// TIA Portal project "weight-based-product-sorting-system" (V16)
// Vorlageprojekt für das Buch mit Zielsystem S7-1200

(* hardware
DEVICE "S7-1200-Station_1"  S7-1200 Station
   slot 0: "Baugruppenträger_0"  Rack  V1.0
   slot 1: "PLC_1"  CPU 1214C DC/DC/DC  6ES7 214-1AG40-0XB0  V4.4
   slot 2: "AQ 4x14BIT_1"  6ES7 232-4HD32-0XB0  V2.1
*)

// ===== PLC "PLC_1"  CPU 1214C DC/DC/DC =====

VAR_GLOBAL   // PLC tag table "Standard-Variablentabelle"
   "Start" AT %I0.0 : Bool;
   "Stop" AT %I0.1 : Bool;
   "Konveyör_Hız_Ayar" AT %IW10 : Int;
   "Giriş_Konveyör" AT %QW20 : Int;
   "Reset_But" AT %I0.2 : Bool;
   "Acil_Stop_But" AT %I0.3 : Bool;
   "Kantar_Giriş_Sensörü" AT %I0.4 : Bool;
   "Kantar_Sensörü" AT %I0.5 : Bool;
   "Kantar_Konveyörü_İleri" AT %Q0.0 : Bool;
   "Ağırlık" AT %IW12 : Int;
   "Transferde_Sensörü" AT %I0.6 : Bool;
   "İleri_Transfer_Konveyörü" AT %Q0.1 : Bool;
   "Ağırlık_Gösterge" AT %QW22 : Int;
   "Sola_Sensör" AT %I0.7 : Bool;
   "Sağa_Sensör" AT %I1.0 : Bool;
   "Sola_Çıkış_Sensörü" AT %I1.1 : Bool;
   "Sağa_Çıkış_Sensörü" AT %I1.2 : Bool;
   "Sağ_Kutu_Sensörü" AT %I1.3 : Bool;
   "Sol_Kutu_Sensörü" AT %I1.4 : Bool;
   "Sol_Konveyör_1" AT %QW24 : Int;
   "Sol_Konveyör_2" AT %Q0.2 : Bool;
   "Sağ_Konveyör_1" AT %QW26 : Int;
   "Sağ_Konveyör_2" AT %Q0.3 : Bool;
   "Sağ_Transfer_Konveyörü" AT %Q0.4 : Bool;
   "Sol_Transfer_Konveyörü" AT %Q0.5 : Bool;
   "Sol_Konveyör_Ürün_Sayısı" AT %QW28 : Int;
   "Sağ_Konveyör_Ürün_Sayısı" AT %QW30 : Int;
   "Alarm" AT %Q0.6 : Bool;
END_VAR

DATA_BLOCK "Memory_Hafıza"   // DB1
{ S7_Optimized_Access := 'TRUE' }
VERSION : 0.1
   VAR
      Sistem_Start : Bool;
      Giriş_Konveyör_Mem : Bool;
      Ağırlık_Tartım : Bool;
      Ağırlık : Int;
      Ağırlık_Mem : Int;
      Sensör_N_Tetik : Bool;
      Kutu_Sensörü_Mem : Bool;
      Sol_Konveyör_Mem : Bool;
      Sol_Transfer_Aktif : Bool;
      Sağ_Transfer_Aktif : Bool;
      Sağ_Konveyör_Mem : Bool;
      Transfer_Mem : Bool;
      Negatif_Kenar : Bool;
      Bekle : Bool;
      Negatif_Kenar_2 : Bool;
      Negatif_Kenar_3 : Bool;
      Negatif_Kenar_4 : Bool;
      Kantar_Hafıza : Bool;
      Ağırlık_Tartım_Pozitif_Kenar : Bool;
      Transfer_Sonlandı : Bool;
      Stop_Hafıza_1 : Bool;
      Negatif_Kenar_5 : Bool;
      Pozitif_Kenar : Bool;
      Interrupt_1 : Int;
      Interrupt_2 : Int;
   END_VAR
BEGIN
END_DATA_BLOCK

DATA_BLOCK "Giriş_Konveyörü_DB1"   // DB2
{ S7_Optimized_Access := 'TRUE' }
VERSION : 0.1
// stored: InstanceOfName Konveyör_Hız
"Konveyör_Hız"
BEGIN
END_DATA_BLOCK

DATA_BLOCK "Sağ_Konveyör"   // DB5
{ S7_Optimized_Access := 'TRUE' }
VERSION : 0.1
// stored: InstanceOfName SAĞ/SOL Konveyör
"SAĞ/SOL Konveyör"
BEGIN
END_DATA_BLOCK

DATA_BLOCK "Sol_Konveyör"   // DB6
{ S7_Optimized_Access := 'TRUE' }
VERSION : 0.1
// stored: InstanceOfName SAĞ/SOL Konveyör
"SAĞ/SOL Konveyör"
BEGIN
END_DATA_BLOCK

DATA_BLOCK "Sol_Konveyör_Hız"   // DB7
{ S7_Optimized_Access := 'TRUE' }
VERSION : 0.1
// stored: InstanceOfName Konveyör_Hız
"Konveyör_Hız"
BEGIN
END_DATA_BLOCK

DATA_BLOCK "Sağ_Konveyör_Hız"   // DB8
{ S7_Optimized_Access := 'TRUE' }
VERSION : 0.1
// stored: InstanceOfName Konveyör_Hız
"Konveyör_Hız"
BEGIN
END_DATA_BLOCK

// folder: System blocks/Program resources

DATA_BLOCK "Timer_1"   // DB3
{ S7_Optimized_Access := 'TRUE' }
AUTHOR : Simatic
FAMILY : IEC
NAME : IEC_TMR
VERSION : 1.0
// stored: InstanceOfName IEC_TIMER
"IEC_TIMER"
BEGIN
END_DATA_BLOCK

DATA_BLOCK "Timer_2"   // DB4
{ S7_Optimized_Access := 'TRUE' }
AUTHOR : Simatic
FAMILY : IEC
NAME : IEC_TMR
VERSION : 1.0
// stored: InstanceOfName IEC_TIMER
"IEC_TIMER"
BEGIN
END_DATA_BLOCK

DATA_BLOCK "Timer_3"   // DB9
{ S7_Optimized_Access := 'TRUE' }
AUTHOR : Simatic
FAMILY : IEC
NAME : IEC_TMR
VERSION : 1.0
// stored: InstanceOfName IEC_TIMER
"IEC_TIMER"
BEGIN
END_DATA_BLOCK

// folder: (top level)

FUNCTION_BLOCK "Konveyör_Hız"   // FB1, LAD
{ S7_Optimized_Access := 'TRUE' }
VERSION : 0.1
   VAR_INPUT
      Konveyör_Hız_Ayar : Int;
      Memory_Hafıza : Bool;
   END_VAR
   VAR_OUTPUT
      Konveyör_Hız : Int;
   END_VAR
BEGIN

REGION Network 1
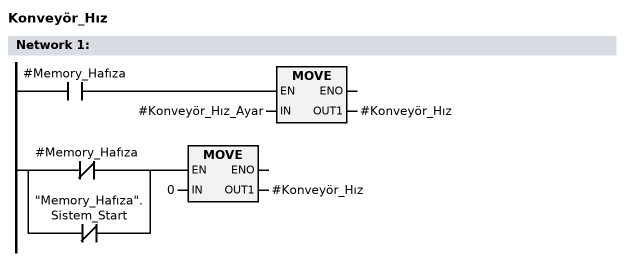
   RUNG wire#powerrail
      Contact( #Memory_Hafıza )
      Move(in := #Konveyör_Hız_Ayar, out1 => #Konveyör_Hız)
   END_RUNG
   RUNG wire#powerrail
      I_Contact( #Memory_Hafıza )
      wire#w1
      Move(in := 0, out1 => #Konveyör_Hız)
   END_RUNG
   RUNG wire#powerrail
      I_Contact( "Memory_Hafıza".Sistem_Start )
   END_RUNG wire#w1
   // the same network as SCL:
   IF #Memory_Hafıza THEN #Konveyör_Hız := #Konveyör_Hız_Ayar; END_IF;
   IF NOT #Memory_Hafıza OR NOT "Memory_Hafıza".Sistem_Start THEN #Konveyör_Hız := 0; END_IF;
END_REGION
END_FUNCTION_BLOCK

FUNCTION_BLOCK "SAĞ/SOL Konveyör"   // FB2, LAD
{ S7_Optimized_Access := 'TRUE' }
VERSION : 0.1
   VAR_INPUT
      Giriş_Sensörü : Bool;
      Çıkış_Sensörü : Bool;
      Kutu_Sensörü : Bool;
      Sayma_Değeri : Int;
   END_VAR
   VAR_OUTPUT
      Aşağı_Konveyör : Bool;
   END_VAR
   VAR_IN_OUT
      Yukarı_Konveyör : Bool;
      Sayma_Degeri_TAM : Bool;
      Ürün_Sayısı : Int;
   END_VAR
   VAR RETAIN
      Counter_Konveyör : CTU_INT;
      Konveyör_Dur : Bool;
   END_VAR
   VAR
      Timer_1 : TON_TIME;
      Konveyör_Devam : Bool;
      Konveyör_Devam_Mem : Bool;
      Timer_2 : TON_TIME;
   END_VAR
BEGIN

REGION Network 1
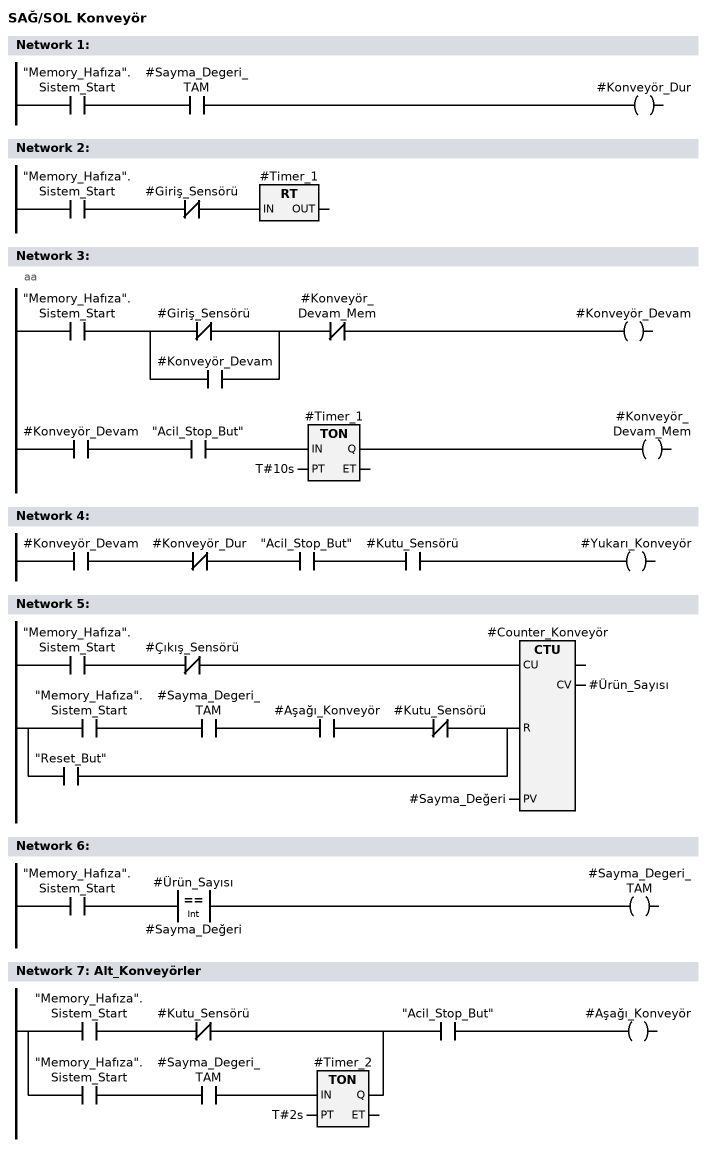
   RUNG wire#powerrail
      Contact( "Memory_Hafıza".Sistem_Start )
      Contact( #Sayma_Degeri_TAM )
      Coil( #Konveyör_Dur )
   END_RUNG
   // the same network as SCL:
   #Konveyör_Dur := "Memory_Hafıza".Sistem_Start AND #Sayma_Degeri_TAM;
END_REGION

REGION Network 2
   RUNG wire#powerrail
      Contact( "Memory_Hafıza".Sistem_Start )
      I_Contact( #Giriş_Sensörü )
      RT_Coil( #Timer_1 )
   END_RUNG
   // the same network as SCL:
   IF "Memory_Hafıza".Sistem_Start AND NOT #Giriş_Sensörü THEN RESET_TIMER(#Timer_1); END_IF;
END_REGION

REGION Network 3
   // aa
   #Konveyör_Devam := "Memory_Hafıza".Sistem_Start AND (NOT #Giriş_Sensörü OR #Konveyör_Devam) AND NOT #Konveyör_Devam_Mem;
   #Timer_1(IN := #Konveyör_Devam AND "Acil_Stop_But", PT := T#10s);   // TON
   #Konveyör_Devam_Mem := #Timer_1.Q;
END_REGION

REGION Network 4
   RUNG wire#powerrail
      Contact( #Konveyör_Devam )
      I_Contact( #Konveyör_Dur )
      Contact( "Acil_Stop_But" )
      Contact( #Kutu_Sensörü )
      Coil( #Yukarı_Konveyör )
   END_RUNG
   // the same network as SCL:
   #Yukarı_Konveyör := #Konveyör_Devam AND NOT #Konveyör_Dur AND "Acil_Stop_But" AND #Kutu_Sensörü;
END_REGION

REGION Network 5
   #Counter_Konveyör(CU := "Memory_Hafıza".Sistem_Start AND NOT #Çıkış_Sensörü,   // CTU
                     R := ("Memory_Hafıza".Sistem_Start AND #Sayma_Degeri_TAM AND #Aşağı_Konveyör AND NOT #Kutu_Sensörü) OR "Reset_But",
                     PV := #Sayma_Değeri,
                     CV => #Ürün_Sayısı);
END_REGION

REGION Network 6
   RUNG wire#powerrail
      Contact( "Memory_Hafıza".Sistem_Start )
      { S7_Templates := "SrcType := Int" } EQ_Contact(in1 := #Ürün_Sayısı, in2 := #Sayma_Değeri)
      Coil( #Sayma_Degeri_TAM )
   END_RUNG
   // the same network as SCL:
   #Sayma_Degeri_TAM := "Memory_Hafıza".Sistem_Start AND (#Ürün_Sayısı = #Sayma_Değeri);
END_REGION

REGION Network 7: Alt_Konveyörler
   #Timer_2(IN := "Memory_Hafıza".Sistem_Start AND #Sayma_Degeri_TAM, PT := T#2s);   // TON
   #Aşağı_Konveyör := (("Memory_Hafıza".Sistem_Start AND NOT #Kutu_Sensörü) OR #Timer_2.Q) AND "Acil_Stop_But";
END_REGION
END_FUNCTION_BLOCK

FUNCTION "MHJ-PLC-Lab-Function-S71200" : Void   // FC9000, SCL
{ S7_Optimized_Access := 'TRUE' }
VERSION : 0.1
   VAR_TEMP
      rdTimeReturn : Int;
      outputTime : DTL;
      SyncVal : Byte;
      forVal : Int;
      forVal_2 : Int;
      Value : Byte;
   END_VAR
   VAR CONSTANT
      CompVal : Byte := 16#34;
      Value_01 : Byte := 16#11;
      Value_01_DW : DWord := 16#A165_D992;
      Value_02_DW : DWord := 16#58BE_4401;
   END_VAR
BEGIN

   #Value:=PEEK(area := 16#82,
        dbNumber := 0,
        byteOffset := 511);
   #Value := #Value + 1;

   POKE(area := 16#82,
        dbNumber := 0,
        byteOffset := 511,
        value := #Value);

   POKE(area:=16#81,
        dbNumber:=0,
        byteOffset:=1016,
        value:=#Value_01_DW);
   POKE(area := 16#81,
        dbNumber := 0,
        byteOffset := 1020,
        value := #Value_02_DW);

   POKE(area := 16#81,
        dbNumber := 0,
        byteOffset := 511,
        value := B#16#00);

   FOR #forVal := 0 TO 120 DO
       FOR #forVal_2:=0 TO 10 DO
           #rdTimeReturn:=RD_SYS_T(#outputTime);
           #rdTimeReturn := WR_SYS_T(#outputTime);
           #rdTimeReturn := RD_SYS_T(#outputTime);
           #rdTimeReturn := WR_SYS_T(#outputTime);
       END_FOR;
       #SyncVal:= PEEK(area := 16#81,
                      dbNumber := 0,
                      byteOffset := 511);
       IF #SyncVal = #CompVal THEN
          GOTO M_1;
       END_IF;
   END_FOR;
   RETURN;

   M_1:
   POKE(area := 16#81,
        dbNumber := 0,
        byteOffset := 511,
        value := B#16#0);
END_FUNCTION

ORGANIZATION_BLOCK "Main"   // OB1, LAD, ProgramCycle
TITLE = "Main Program Sweep (Cycle)"
{ S7_Optimized_Access := 'TRUE' }
VERSION : 0.1
   VAR_INPUT
      Initial_Call : Bool;   // Initial call of this OB
      Remanence : Bool;   // =True, if remanent data are available
   END_VAR
   VAR_TEMP   // added for the SCL form of the ladder/FBD networks
      _w1 : Bool;
      _w2 : Bool;
   END_VAR
BEGIN

REGION Network 1: Konnektierungsbaustein für PLC-Lab
   // Im Netzwerk 1 wird der Konnektierungsbaustein für PLC-Lab aufgerufen.
   // Dieser Aufruf darf nicht entfernt werden!
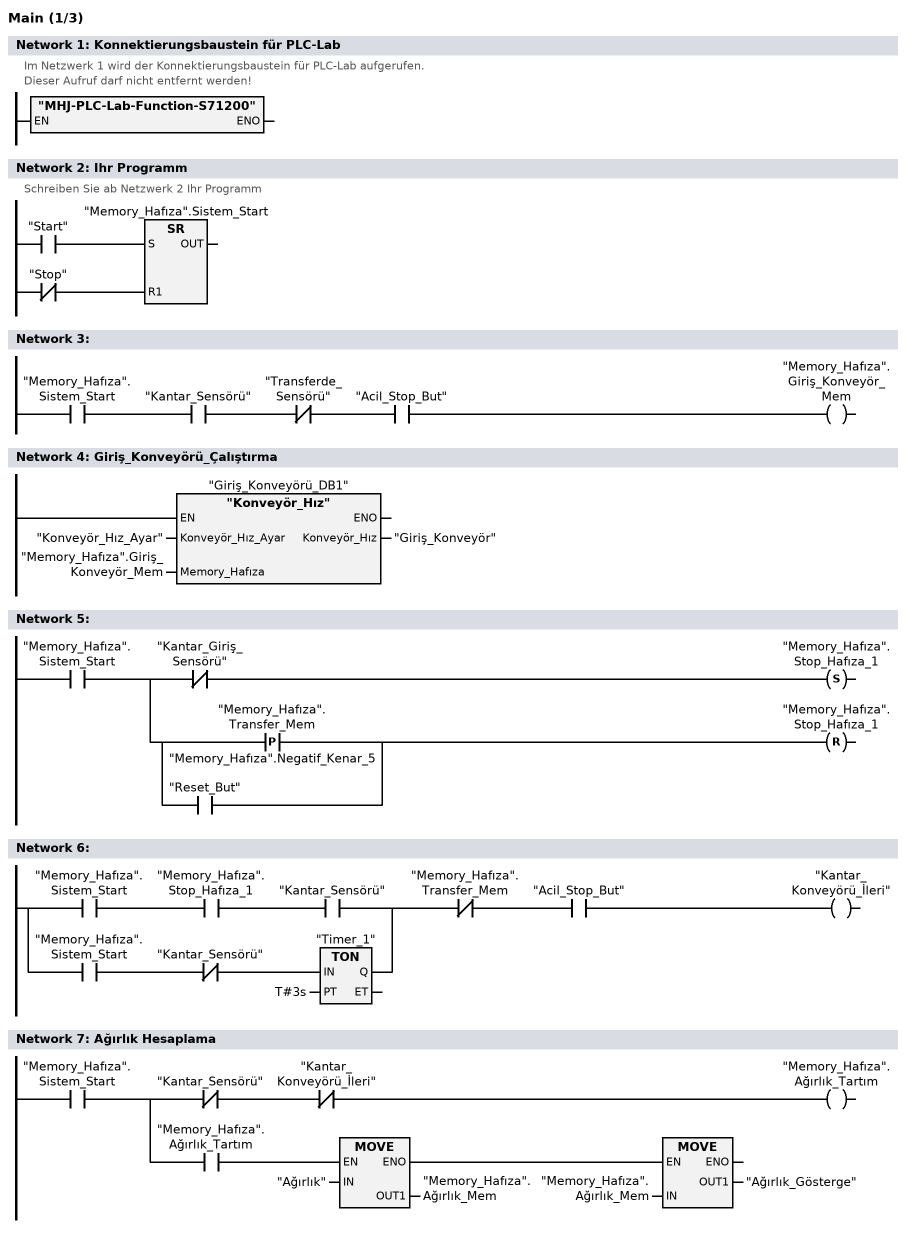
   RUNG wire#powerrail
      "MHJ-PLC-Lab-Function-S71200"()
   END_RUNG
   // the same network as SCL:
   "MHJ-PLC-Lab-Function-S71200"();
END_REGION

REGION Network 2: Ihr Programm
   // Schreiben Sie ab Netzwerk 2 Ihr Programm
   RUNG wire#powerrail
      Contact( "Start" )
      S_SR(operand := "Memory_Hafıza".Sistem_Start, r1 := wire#w1)
   END_RUNG
   RUNG wire#powerrail
      I_Contact( "Stop" )
   END_RUNG wire#w1
   // the same network as SCL:
   IF "Start" THEN
       "Memory_Hafıza".Sistem_Start := TRUE;   // SR flip-flop
   END_IF;
   IF NOT "Stop" THEN "Memory_Hafıza".Sistem_Start := FALSE; END_IF;
END_REGION

REGION Network 3
   RUNG wire#powerrail
      Contact( "Memory_Hafıza".Sistem_Start )
      Contact( "Kantar_Sensörü" )
      I_Contact( "Transferde_Sensörü" )
      Contact( "Acil_Stop_But" )
      Coil( "Memory_Hafıza".Giriş_Konveyör_Mem )
   END_RUNG
   // the same network as SCL:
   "Memory_Hafıza".Giriş_Konveyör_Mem := "Memory_Hafıza".Sistem_Start AND "Kantar_Sensörü" AND NOT "Transferde_Sensörü" AND "Acil_Stop_But";
END_REGION

REGION Network 4: Giriş_Konveyörü_Çalıştırma
   RUNG wire#powerrail
      "Giriş_Konveyörü_DB1"(Konveyör_Hız_Ayar := "Konveyör_Hız_Ayar", Memory_Hafıza := "Memory_Hafıza".Giriş_Konveyör_Mem, Konveyör_Hız => "Giriş_Konveyör")
   END_RUNG
   // the same network as SCL:
   "Giriş_Konveyörü_DB1"(Konveyör_Hız_Ayar := "Konveyör_Hız_Ayar",   // "Konveyör_Hız"
                         Memory_Hafıza := "Memory_Hafıza".Giriş_Konveyör_Mem,
                         Konveyör_Hız => "Giriş_Konveyör");
END_REGION

REGION Network 5
   RUNG wire#powerrail
      Contact( "Memory_Hafıza".Sistem_Start )
      wire#w1
      I_Contact( "Kantar_Giriş_Sensörü" )
      S_Coil( "Memory_Hafıza".Stop_Hafıza_1 )
   END_RUNG
   RUNG wire#w1
      P_Contact(operand := "Memory_Hafıza".Transfer_Mem, bit := "Memory_Hafıza".Negatif_Kenar_5)
      wire#w2
      R_Coil( "Memory_Hafıza".Stop_Hafıza_1 )
   END_RUNG
   RUNG wire#w1
      Contact( "Reset_But" )
   END_RUNG wire#w2
   // the same network as SCL:
   IF "Memory_Hafıza".Sistem_Start AND NOT "Kantar_Giriş_Sensörü" THEN
       "Memory_Hafıza".Stop_Hafıza_1 := TRUE;
   END_IF;
   #_w1 := "Memory_Hafıza".Sistem_Start AND "Memory_Hafıza".Transfer_Mem AND NOT "Memory_Hafıza".Negatif_Kenar_5;   // rising edge of "Memory_Hafıza".Transfer_Mem
   "Memory_Hafıza".Negatif_Kenar_5 := "Memory_Hafıza".Transfer_Mem;
   IF #_w1 OR ("Memory_Hafıza".Sistem_Start AND "Reset_But") THEN
       "Memory_Hafıza".Stop_Hafıza_1 := FALSE;
   END_IF;
END_REGION

REGION Network 6
   "Timer_1".TON(IN := "Memory_Hafıza".Sistem_Start AND NOT "Kantar_Sensörü", PT := T#3s);
   "Kantar_Konveyörü_İleri" := (("Memory_Hafıza".Sistem_Start AND "Memory_Hafıza".Stop_Hafıza_1 AND "Kantar_Sensörü") OR "Timer_1".Q) AND NOT "Memory_Hafıza".Transfer_Mem AND "Acil_Stop_But";
END_REGION

REGION Network 7: Ağırlık Hesaplama
   RUNG wire#powerrail
      Contact( "Memory_Hafıza".Sistem_Start )
      wire#w1
      I_Contact( "Kantar_Sensörü" )
      I_Contact( "Kantar_Konveyörü_İleri" )
      Coil( "Memory_Hafıza".Ağırlık_Tartım )
   END_RUNG
   RUNG wire#w1
      Contact( "Memory_Hafıza".Ağırlık_Tartım )
      Move(in := "Ağırlık", out1 => "Memory_Hafıza".Ağırlık_Mem)
      Move(in := "Memory_Hafıza".Ağırlık_Mem, out1 => "Ağırlık_Gösterge")
   END_RUNG
   // the same network as SCL:
   "Memory_Hafıza".Ağırlık_Tartım := "Memory_Hafıza".Sistem_Start AND NOT "Kantar_Sensörü" AND NOT "Kantar_Konveyörü_İleri";
   IF "Memory_Hafıza".Sistem_Start AND "Memory_Hafıza".Ağırlık_Tartım THEN
       "Memory_Hafıza".Ağırlık_Mem := "Ağırlık";
       "Ağırlık_Gösterge" := "Memory_Hafıza".Ağırlık_Mem;
   END_IF;
END_REGION

REGION Network 8
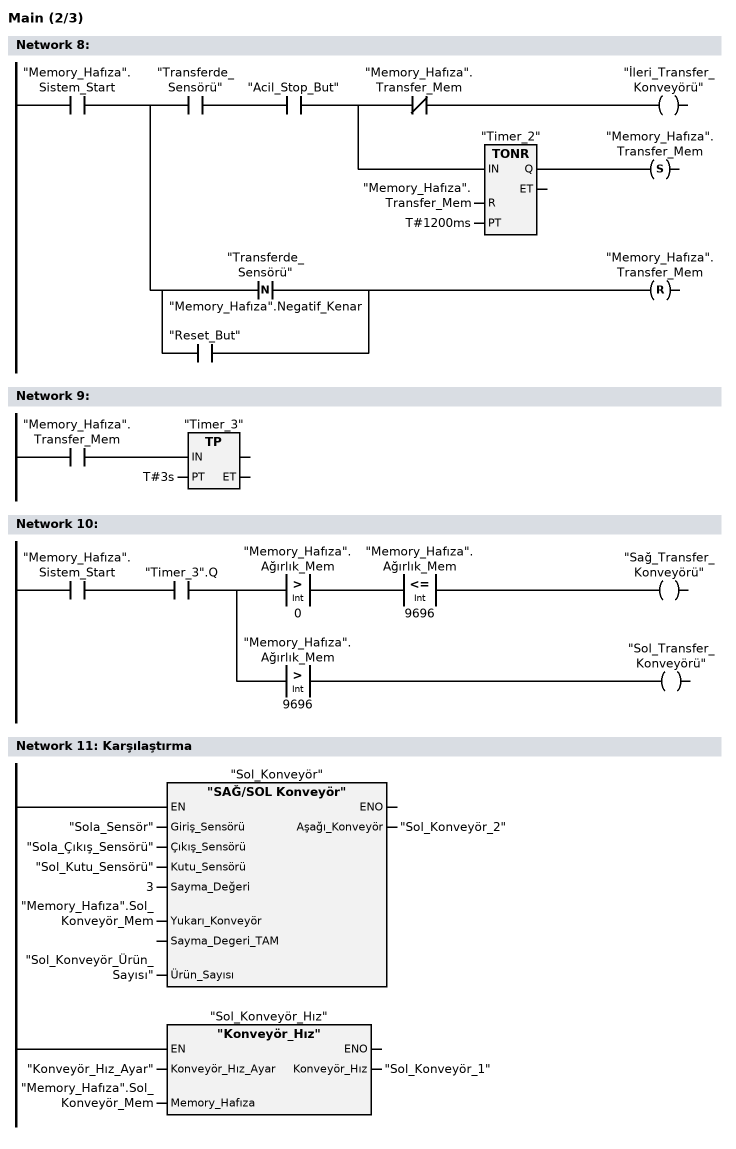
   #_w1 := "Memory_Hafıza".Sistem_Start AND "Transferde_Sensörü" AND "Acil_Stop_But";
   "İleri_Transfer_Konveyörü" := #_w1 AND NOT "Memory_Hafıza".Transfer_Mem;
   "Timer_2".TONR(IN := #_w1, R := "Memory_Hafıza".Transfer_Mem, PT := T#1200ms);
   IF "Timer_2".Q THEN "Memory_Hafıza".Transfer_Mem := TRUE; END_IF;
   #_w2 := "Memory_Hafıza".Sistem_Start AND NOT "Transferde_Sensörü" AND "Memory_Hafıza".Negatif_Kenar;   // falling edge of "Transferde_Sensörü"
   "Memory_Hafıza".Negatif_Kenar := "Transferde_Sensörü";
   IF #_w2 OR ("Memory_Hafıza".Sistem_Start AND "Reset_But") THEN
       "Memory_Hafıza".Transfer_Mem := FALSE;
   END_IF;
END_REGION

REGION Network 9
   "Timer_3".TP(IN := "Memory_Hafıza".Transfer_Mem, PT := T#3s);
END_REGION

REGION Network 10
   RUNG wire#powerrail
      Contact( "Memory_Hafıza".Sistem_Start )
      Contact( "Timer_3".Q )
      wire#w1
      { S7_Templates := "SrcType := Int" } GT_Contact(in1 := "Memory_Hafıza".Ağırlık_Mem, in2 := 0)
      { S7_Templates := "SrcType := Int" } LE_Contact(in1 := "Memory_Hafıza".Ağırlık_Mem, in2 := 9696)
      Coil( "Sağ_Transfer_Konveyörü" )
   END_RUNG
   RUNG wire#w1
      { S7_Templates := "SrcType := Int" } GT_Contact(in1 := "Memory_Hafıza".Ağırlık_Mem, in2 := 9696)
      Coil( "Sol_Transfer_Konveyörü" )
   END_RUNG
   // the same network as SCL:
   #_w1 := "Memory_Hafıza".Sistem_Start AND "Timer_3".Q;
   "Sağ_Transfer_Konveyörü" := #_w1 AND ("Memory_Hafıza".Ağırlık_Mem > 0) AND ("Memory_Hafıza".Ağırlık_Mem <= 9696);
   "Sol_Transfer_Konveyörü" := #_w1 AND ("Memory_Hafıza".Ağırlık_Mem > 9696);
END_REGION

REGION Network 11: Karşılaştırma
   RUNG wire#powerrail
      "Sol_Konveyör"(Giriş_Sensörü := "Sola_Sensör", Çıkış_Sensörü := "Sola_Çıkış_Sensörü", Kutu_Sensörü := "Sol_Kutu_Sensörü", Sayma_Değeri := 3, Yukarı_Konveyör := "Memory_Hafıza".Sol_Konveyör_Mem, Sayma_Degeri_TAM :=, Ürün_Sayısı := "Sol_Konveyör_Ürün_Sayısı", Aşağı_Konveyör => "Sol_Konveyör_2")
   END_RUNG
   RUNG wire#powerrail
      "Sol_Konveyör_Hız"(Konveyör_Hız_Ayar := "Konveyör_Hız_Ayar", Memory_Hafıza := "Memory_Hafıza".Sol_Konveyör_Mem, Konveyör_Hız => "Sol_Konveyör_1")
   END_RUNG
   // the same network as SCL:
   "Sol_Konveyör"(Giriş_Sensörü := "Sola_Sensör",   // "SAĞ/SOL Konveyör"
                  Çıkış_Sensörü := "Sola_Çıkış_Sensörü",
                  Kutu_Sensörü := "Sol_Kutu_Sensörü",
                  Sayma_Değeri := 3,
                  Yukarı_Konveyör := "Memory_Hafıza".Sol_Konveyör_Mem,
                  Ürün_Sayısı := "Sol_Konveyör_Ürün_Sayısı",
                  Aşağı_Konveyör => "Sol_Konveyör_2");
   "Sol_Konveyör_Hız"(Konveyör_Hız_Ayar := "Konveyör_Hız_Ayar",   // "Konveyör_Hız"
                      Memory_Hafıza := "Memory_Hafıza".Sol_Konveyör_Mem,
                      Konveyör_Hız => "Sol_Konveyör_1");
END_REGION

REGION Network 12
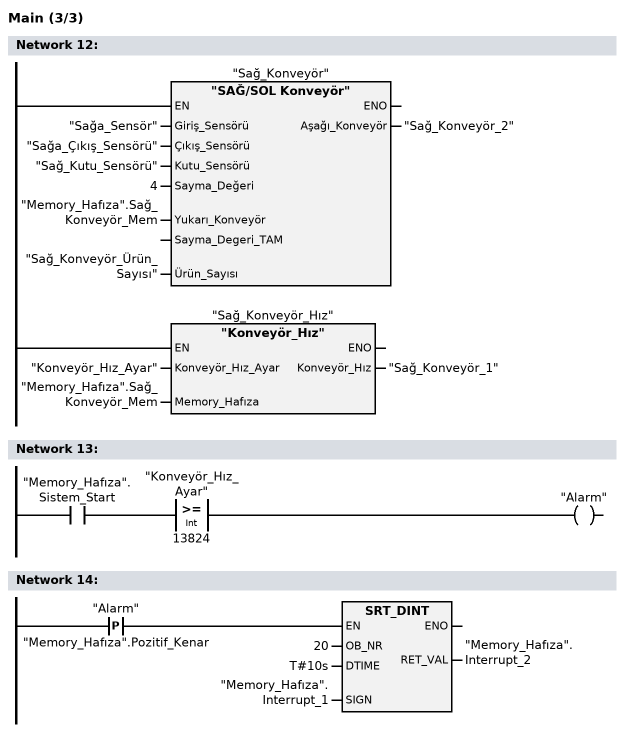
   RUNG wire#powerrail
      "Sağ_Konveyör"(Giriş_Sensörü := "Sağa_Sensör", Çıkış_Sensörü := "Sağa_Çıkış_Sensörü", Kutu_Sensörü := "Sağ_Kutu_Sensörü", Sayma_Değeri := 4, Yukarı_Konveyör := "Memory_Hafıza".Sağ_Konveyör_Mem, Sayma_Degeri_TAM :=, Ürün_Sayısı := "Sağ_Konveyör_Ürün_Sayısı", Aşağı_Konveyör => "Sağ_Konveyör_2")
   END_RUNG
   RUNG wire#powerrail
      "Sağ_Konveyör_Hız"(Konveyör_Hız_Ayar := "Konveyör_Hız_Ayar", Memory_Hafıza := "Memory_Hafıza".Sağ_Konveyör_Mem, Konveyör_Hız => "Sağ_Konveyör_1")
   END_RUNG
   // the same network as SCL:
   "Sağ_Konveyör"(Giriş_Sensörü := "Sağa_Sensör",   // "SAĞ/SOL Konveyör"
                  Çıkış_Sensörü := "Sağa_Çıkış_Sensörü",
                  Kutu_Sensörü := "Sağ_Kutu_Sensörü",
                  Sayma_Değeri := 4,
                  Yukarı_Konveyör := "Memory_Hafıza".Sağ_Konveyör_Mem,
                  Ürün_Sayısı := "Sağ_Konveyör_Ürün_Sayısı",
                  Aşağı_Konveyör => "Sağ_Konveyör_2");
   "Sağ_Konveyör_Hız"(Konveyör_Hız_Ayar := "Konveyör_Hız_Ayar",   // "Konveyör_Hız"
                      Memory_Hafıza := "Memory_Hafıza".Sağ_Konveyör_Mem,
                      Konveyör_Hız => "Sağ_Konveyör_1");
END_REGION

REGION Network 13
   RUNG wire#powerrail
      Contact( "Memory_Hafıza".Sistem_Start )
      { S7_Templates := "SrcType := Int" } GE_Contact(in1 := "Konveyör_Hız_Ayar", in2 := 13824)
      Coil( "Alarm" )
   END_RUNG
   // the same network as SCL:
   "Alarm" := "Memory_Hafıza".Sistem_Start AND ("Konveyör_Hız_Ayar" >= 13824);
END_REGION

REGION Network 14
   #_w1 := "Alarm" AND NOT "Memory_Hafıza".Pozitif_Kenar;   // rising edge of "Alarm"
   "Memory_Hafıza".Pozitif_Kenar := "Alarm";
   IF #_w1 THEN
       "Memory_Hafıza".Interrupt_2 := SRT_DINT(OB_NR := 20, DTIME := T#10s, SIGN := "Memory_Hafıza".Interrupt_1);
   END_IF;
END_REGION
END_ORGANIZATION_BLOCK

ORGANIZATION_BLOCK "Time delay interrupt"   // OB20, LAD, TimeDelayInterrupt
{ S7_Optimized_Access := 'TRUE' }
VERSION : 0.1
   VAR_INPUT
      Sign : Word;   // Identifier input (SIGN) passed to triggering call of SRT_DINT
   END_VAR
BEGIN

REGION Network 1
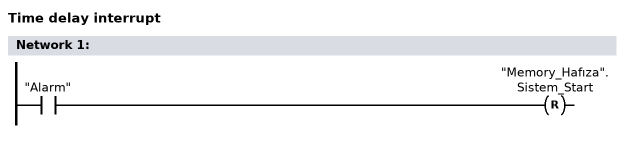
   RUNG wire#powerrail
      Contact( "Alarm" )
      R_Coil( "Memory_Hafıza".Sistem_Start )
   END_RUNG
   // the same network as SCL:
   IF "Alarm" THEN "Memory_Hafıza".Sistem_Start := FALSE; END_IF;
END_REGION
END_ORGANIZATION_BLOCK